// TIA Portal V17 export
// export: Created 2025-03-05T07:59:14.198006Z, ExportSetting WithDefaults, DisplayName Totally Integrated Automation Portal, DisplayVersion V17 Update 8, DisplayName TIA Portal Openness, DisplayVersion V17 Update 8, DisplayName TIA Portal Version Control Interface, DisplayVersion V17, DisplayName SINAMICS Startdrive Advanced, DisplayVersion V17 SP2, DisplayName SINAMICS Startdrive G110M, G120, G120C, G120D, G120P, G115D, DisplayVersion V17 SP2, DisplayName SINAMICS Startdrive G130, G150, S120, S150, SINAMICS MV, S210, DisplayVersion V17 SP2, DisplayName STEP 7 Professional, DisplayVersion V17 Update 8, DisplayName SINUMERIK ONE STEP 7 Toolbox, DisplayVersion V17 Update 12, DisplayName SINUMERIK 840D sl STEP 7 Toolbox, DisplayVersion V17 Update 12, DisplayName STEP 7 Safety, DisplayVersion V17 Update 6, DisplayName WinCC Advanced, DisplayVersion V17 Update 8
DATA_BLOCK "DB4000_FIX_TABLE_POSITIONS"   // DB4000
{ S7_Optimized_Access := 'FALSE'; DB_Accessible_From_OPC_UA := 'FALSE' }
AUTHOR : ETXETAR
VERSION : 1.0
// stored: AutoNumber false, DBAccessibleFromOPCUA false, DBAccessibleFromWebserver true, IsOnlyStoredInLoadMemory false, IsWriteProtectedInAS false
   VAR RETAIN
      UNIT_01 : Struct
         FIXTURE_1 : Struct
            IN_LOAD_UNLOAD_STATION_1 : Bool;   // UNIT 01 FIXTURE 1 IN LOAD UNLOAD STATION
            IN_SPARE_STATION_2 : Bool;   // UNIT 01 FIXTURE 1 IN SPARE STATION
            IN_CLADDING_STATION_3 : Bool;   // UNIT 01 FIXTURE 1 IN CLADDING STATION
            IN_CLEAN_STATION_4 : Bool;   // UNIT 01 FIXTURE 1 IN CLEANING STATION
            NO_DEFINED_POSITION : Bool;   // UNIT 01 FIXTURE 1 IN NO DEFINED POSITION
         END_STRUCT;
         FIXTURE_2 : Struct
            IN_LOAD_UNLOAD_STATION_1 : Bool;   // UNIT 01 FIXTURE 2 IN LOAD UNLOAD STATION
            IN_SPARE_STATION_2 : Bool;   // UNIT 01 FIXTURE 2 IN SPARE STATION
            IN_CLADDING_STATION_3 : Bool;   // UNIT 01 FIXTURE 2 IN CLADDING STATION
            IN_CLEAN_STATION_4 : Bool;   // UNIT 01 FIXTURE 2 IN CLEANING STATION
            NO_DEFINED_POSITION : Bool;   // UNIT 01 FIXTURE 2 IN NO DEFINED POSITION
         END_STRUCT;
         FIXTURE_3 : Struct
            IN_LOAD_UNLOAD_STATION_1 : Bool;   // UNIT 01 FIXTURE 3 IN LOAD UNLOAD STATION
            IN_SPARE_STATION_2 : Bool;   // UNIT 01 FIXTURE 3 IN SPARE STATION
            IN_CLADDING_STATION_3 : Bool;   // UNIT 01 FIXTURE 3 IN CLADDING STATION
            IN_CLEAN_STATION_4 : Bool;   // UNIT 01 FIXTURE 3 IN CLEANING STATION
            NO_DEFINED_POSITION : Bool;   // UNIT 01 FIXTURE 3 IN NO DEFINED POSITION
         END_STRUCT;
         FIXTURE_4 : Struct
            IN_LOAD_UNLOAD_STATION_1 : Bool;   // UNIT 01 FIXTURE 4 IN LOAD UNLOAD STATION
            IN_SPARE_STATION_2 : Bool;   // UNIT 01 FIXTURE 4 IN SPARE STATION
            IN_CLADDING_STATION_3 : Bool;   // UNIT 01 FIXTURE 4 IN CLADDING STATION
            IN_CLEAN_STATION_4 : Bool;   // UNIT 01 FIXTURE 4 IN CLEANING STATION
            NO_DEFINED_POSITION : Bool;   // UNIT 01 FIXTURE 4 IN NO DEFINED POSITION
         END_STRUCT;
         AXIS_E10_HOME_POS : Bool;   // AXIS E10 IN HOME POSITION
         AXIS_E10_NOT_DEFINED_POS : Bool;   // AXIS E10 NOT IN A DEFINED POSITION
         SPARE : UInt;   // AXIS E10 POSITION SENSOR VALUE
         E10_POSITION_REACH : Struct
            E10_0_DEGREES : Bool;   // E10 AXIS 0 DEGREES POSITION REACH
            E10_90_DEGREES : Bool;   // E10 AXIS 90 DEGREES POSITION REACH
            E10_180_DEGREES : Bool;   // E10 AXIS 180 DEGREES POSITION REACH
            E10_270_DEGREES : Bool;   // E10 AXIS 270 DEGREES POSITION REACH
            E10_0_DEGREES_FLANGE : Bool;   // E10 AXIS 0 DEGREES POSITION REACH FLANGE
            E10_90_DEGREES_FLANGE : Bool;   // E10 AXIS 90 DEGREES POSITION REACH FLANGE
            E10_180_DEGREES_FLANGE : Bool;   // E10 AXIS 180 DEGREES POSITION REACH FLANGE
            E10_270_DEGREES_FLANGE : Bool;   // E10 AXIS 270 DEGREES POSITION REACH FLANGE
         END_STRUCT;
         FIXTURE_NUMBER_IN : Struct
            STATION_1 : Int;   // FIXTURE NUMBER IN STATION 1
            STATION_2 : Int;   // FIXTURE NUMBER IN STATION 2
            STATION_3 : Int;   // FIXTURE NUMBER IN STATION 3
            STATION_4 : Int;   // FIXTURE NUMBER IN STATION 4
         END_STRUCT;
      END_STRUCT;
      UNIT_02 : Struct
         FIXTURE_1 : Struct
            IN_LOAD_UNLOAD_STATION_1 : Bool;   // UNIT 02 FIXTURE 1 IN LOAD UNLOAD STATION
            IN_MEASURING_STATION_2 : Bool;   // UNIT 02 FIXTURE 1 IN SPARE STATION
            IN_CLADDING_STATION_3 : Bool;   // UNIT 02 FIXTURE 1 IN CLADDING STATION
            IN_CLEAN_STATION_4 : Bool;   // UNIT 02 FIXTURE 1 IN MEASURING/CLEANING STATION
            NO_DEFINED_POSITION : Bool;   // UNIT 02 FIXTURE 1 IN NO DEFINED POSITION
         END_STRUCT;
         FIXTURE_2 : Struct
            IN_LOAD_UNLOAD_STATION_1 : Bool;   // UNIT 02 FIXTURE 2 IN LOAD UNLOAD STATION
            IN_MEASURING_STATION_2 : Bool;   // UNIT 02 FIXTURE 2 IN SPARE STATION
            IN_CLADDING_STATION_3 : Bool;   // UNIT 02 FIXTURE 2 IN CLADDING STATION
            IN_CLEAN_STATION_4 : Bool;   // UNIT 02 FIXTURE 2 IN MEASURING/CLEANING STATION
            NO_DEFINED_POSITION : Bool;   // UNIT 02 FIXTURE 2 IN NO DEFINED POSITION
         END_STRUCT;
         FIXTURE_3 : Struct
            IN_LOAD_UNLOAD_STATION_1 : Bool;   // UNIT 02 FIXTURE 3 IN LOAD UNLOAD STATION
            IN_MEASURING_STATION_2 : Bool;   // UNIT 02 FIXTURE 3 IN SPARE STATION
            IN_CLADDING_STATION_3 : Bool;   // UNIT 02 FIXTURE 3 IN CLADDING STATION
            IN_CLEAN_STATION_4 : Bool;   // UNIT 02 FIXTURE 3 IN MEASURING/CLEANING STATION
            NO_DEFINED_POSITION : Bool;   // UNIT 02 FIXTURE 3 IN NO DEFINED POSITION
         END_STRUCT;
         FIXTURE_4 : Struct
            IN_LOAD_UNLOAD_STATION_1 : Bool;   // UNIT 02 FIXTURE 4 IN LOAD UNLOAD STATION
            IN_MEASURING_STATION_2 : Bool;   // UNIT 02 FIXTURE 4 IN SPARE STATION
            IN_CLADDING_STATION_3 : Bool;   // UNIT 02 FIXTURE 4 IN CLADDING STATION
            IN_CLEAN_STATION_4 : Bool;   // UNIT 02 FIXTURE 4 IN MEASURING/CLEANING STATION
            NO_DEFINED_POSITION : Bool;   // UNIT 02 FIXTURE 4 IN NO DEFINED POSITION
         END_STRUCT;
         AXIS_E20_HOME_POS : Bool;   // AXIS E20 IN HOME POSITION
         AXIS_E20_NOT_DEFINED_POS : Bool;   // AXIS E20 NOT IN A DEFINED POSITION
         SPARE : UInt;   // E20 POSITION SENSOR VALUE
         E20_POSITION_REACH : Struct
            E20_0_DEGREES : Bool;   // E20 AXIS 0 DEGREES POSITION REACH
            E20_90_DEGREES : Bool;   // E20 AXIS 90 DEGREES POSITION REACH
            E20_180_DEGREES : Bool;   // E20 AXIS 180 DEGREES POSITION REACH
            E20_270_DEGREES : Bool;   // E20 AXIS 270 DEGREES POSITION REACH
            E20_0_DEGREES_FLANGE : Bool;   // E20 AXIS 0 DEGREES POSITION REACH FLANGE
            E20_90_DEGREES_FLANGE : Bool;   // E20 AXIS 90 DEGREES POSITION REACH FLANGE
            E20_180_DEGREES_FLANGE : Bool;   // E20 AXIS 180 DEGREES POSITION REACH FLANGE
            E20_270_DEGREES_FLANGE : Bool;   // E20 AXIS 270 DEGREES POSITION REACH FLANGE
         END_STRUCT;
         FIXTURE_NUMBER_IN : Struct
            STATION_1 : Int;   // FIXTURE NUMBER IN STATION 1
            STATION_2 : Int;   // FIXTURE NUMBER IN STATION 2
            STATION_3 : Int;   // FIXTURE NUMBER IN STATION 3
            STATION_4 : Int;   // FIXTURE NUMBER IN STATION 4
         END_STRUCT;
      END_STRUCT;
   END_VAR
BEGIN
END_DATA_BLOCK
